// TIA Portal V17 export
// export: Created 2023-12-22T15:04:43.0097959Z, ExportSetting WithDefaults, DisplayName Totally Integrated Automation Portal, DisplayVersion V17, DisplayName TIA Portal Openness, DisplayVersion V17, DisplayName TIA Portal Version Control Interface, DisplayVersion V17, DisplayName STEP 7 Professional, DisplayVersion V17, DisplayName STEP 7 Safety, DisplayVersion V17, DisplayName WinCC Advanced, DisplayVersion V17
FUNCTION "drv_Mode" : Void   // FC150, LAD
{ S7_Optimized_Access := 'FALSE' }
VERSION : 0.1
// stored: AutoNumber false, IsIECCheckEnabled false, SetENOAutomatically false, UDAEnableTagReadback false
   VAR_INPUT
      CMD : "CMD";   // Основные команды / Блок команд
      All_Block : Bool;   // Аварийная блокировка
   END_VAR
   VAR_OUTPUT
      Mode : Int;   // Режим работы
   END_VAR
BEGIN

REGION Network 1: Автоматический режим
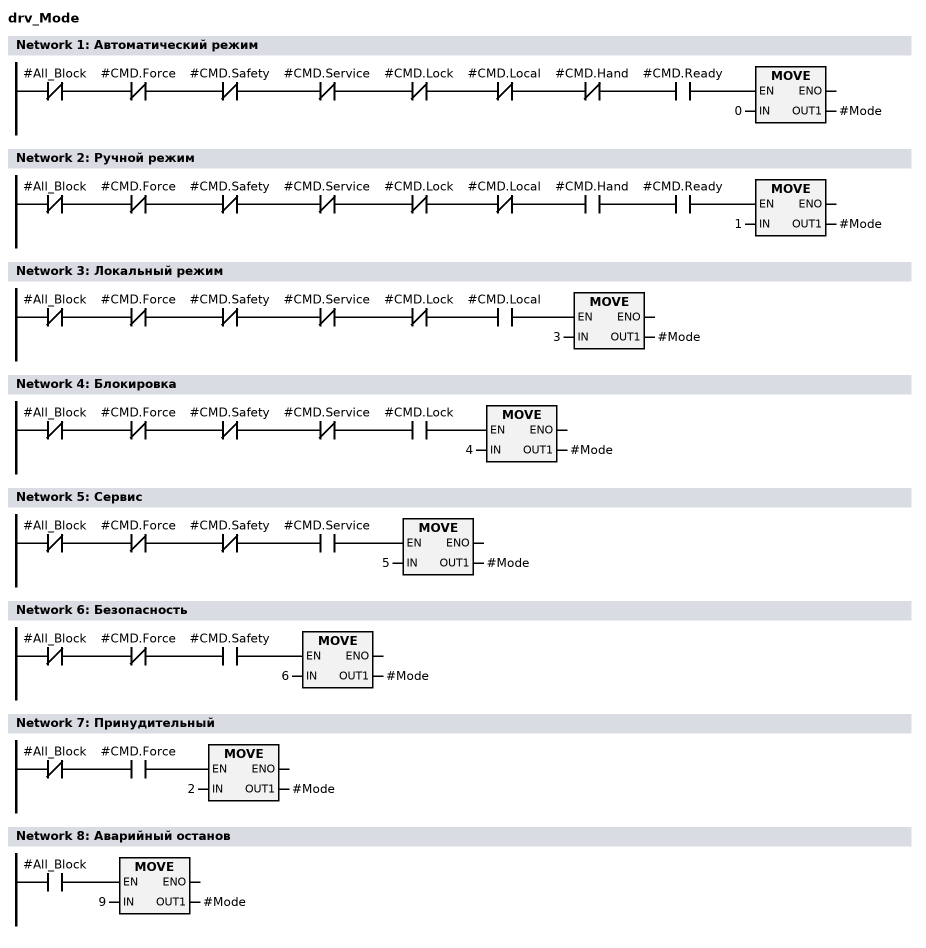
   RUNG wire#powerrail
      I_Contact( #All_Block )
      I_Contact( #CMD.Force )
      I_Contact( #CMD.Safety )
      I_Contact( #CMD.Service )
      I_Contact( #CMD.Lock )
      I_Contact( #CMD.Local )
      I_Contact( #CMD.Hand )
      Contact( #CMD.Ready )
      { S7_GenerateENO := "TRUE" } Move(in := 0, out1 => #Mode)
   END_RUNG
   // the same network as SCL:
   IF NOT #All_Block AND NOT #CMD.Force AND NOT #CMD.Safety AND NOT #CMD.Service AND NOT #CMD.Lock AND NOT #CMD.Local AND NOT #CMD.Hand AND #CMD.Ready THEN
       #Mode := 0;
   END_IF;
END_REGION

REGION Network 2: Ручной режим
   RUNG wire#powerrail
      I_Contact( #All_Block )
      I_Contact( #CMD.Force )
      I_Contact( #CMD.Safety )
      I_Contact( #CMD.Service )
      I_Contact( #CMD.Lock )
      I_Contact( #CMD.Local )
      Contact( #CMD.Hand )
      Contact( #CMD.Ready )
      { S7_GenerateENO := "TRUE" } Move(in := 1, out1 => #Mode)
   END_RUNG
   // the same network as SCL:
   IF NOT #All_Block AND NOT #CMD.Force AND NOT #CMD.Safety AND NOT #CMD.Service AND NOT #CMD.Lock AND NOT #CMD.Local AND #CMD.Hand AND #CMD.Ready THEN
       #Mode := 1;
   END_IF;
END_REGION

REGION Network 3: Локальный режим
   RUNG wire#powerrail
      I_Contact( #All_Block )
      I_Contact( #CMD.Force )
      I_Contact( #CMD.Safety )
      I_Contact( #CMD.Service )
      I_Contact( #CMD.Lock )
      Contact( #CMD.Local )
      { S7_GenerateENO := "TRUE" } Move(in := 3, out1 => #Mode)
   END_RUNG
   // the same network as SCL:
   IF NOT #All_Block AND NOT #CMD.Force AND NOT #CMD.Safety AND NOT #CMD.Service AND NOT #CMD.Lock AND #CMD.Local THEN
       #Mode := 3;
   END_IF;
END_REGION

REGION Network 4: Блокировка
   RUNG wire#powerrail
      I_Contact( #All_Block )
      I_Contact( #CMD.Force )
      I_Contact( #CMD.Safety )
      I_Contact( #CMD.Service )
      Contact( #CMD.Lock )
      { S7_GenerateENO := "TRUE" } Move(in := 4, out1 => #Mode)
   END_RUNG
   // the same network as SCL:
   IF NOT #All_Block AND NOT #CMD.Force AND NOT #CMD.Safety AND NOT #CMD.Service AND #CMD.Lock THEN
       #Mode := 4;
   END_IF;
END_REGION

REGION Network 5: Сервис
   RUNG wire#powerrail
      I_Contact( #All_Block )
      I_Contact( #CMD.Force )
      I_Contact( #CMD.Safety )
      Contact( #CMD.Service )
      { S7_GenerateENO := "TRUE" } Move(in := 5, out1 => #Mode)
   END_RUNG
   // the same network as SCL:
   IF NOT #All_Block AND NOT #CMD.Force AND NOT #CMD.Safety AND #CMD.Service THEN #Mode := 5; END_IF;
END_REGION

REGION Network 6: Безопасность
   RUNG wire#powerrail
      I_Contact( #All_Block )
      I_Contact( #CMD.Force )
      Contact( #CMD.Safety )
      { S7_GenerateENO := "TRUE" } Move(in := 6, out1 => #Mode)
   END_RUNG
   // the same network as SCL:
   IF NOT #All_Block AND NOT #CMD.Force AND #CMD.Safety THEN #Mode := 6; END_IF;
END_REGION

REGION Network 7: Принудительный
   RUNG wire#powerrail
      I_Contact( #All_Block )
      Contact( #CMD.Force )
      { S7_GenerateENO := "TRUE" } Move(in := 2, out1 => #Mode)
   END_RUNG
   // the same network as SCL:
   IF NOT #All_Block AND #CMD.Force THEN #Mode := 2; END_IF;
END_REGION

REGION Network 8: Аварийный останов
   RUNG wire#powerrail
      Contact( #All_Block )
      { S7_GenerateENO := "TRUE" } Move(in := 9, out1 => #Mode)
   END_RUNG
   // the same network as SCL:
   IF #All_Block THEN #Mode := 9; END_IF;
END_REGION
END_FUNCTION
